TYPE "TExtEncoder_StatusWord"
VERSION : 0.1
// Block: TExtEncoder_StatusWord
   STRUCT
      Enable : Bool;
      Error : Bool;
      RestartActive : Bool;
      OnlineStartValuesChanged : Bool;
      HomingDone : Bool;
      Done : Bool;
      HomingCommand : Bool;
   END_STRUCT;

END_TYPE
